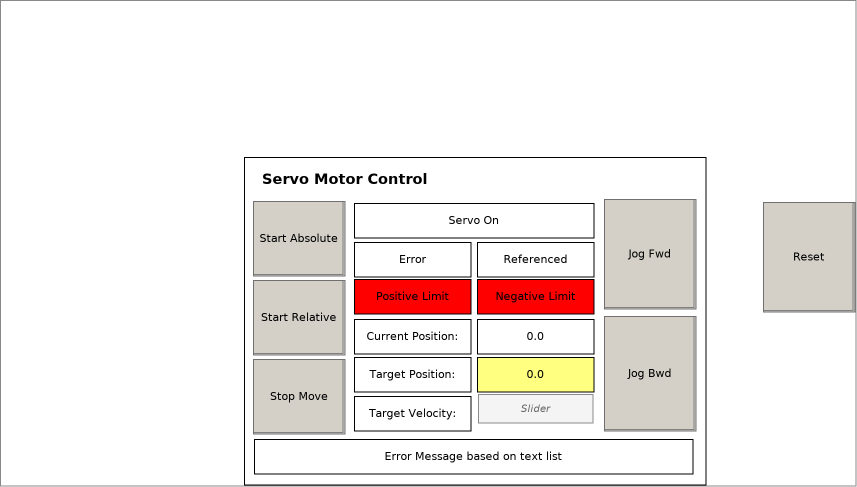
VISUALIZATION Std_BoschServo_Ctrl  // 857x487
    Rectangle (244,157 462x328)
    Button (604,199 92x110), "Jog Fwd"
        tap ER_Arm_Srv_Var.In_JogFwd
    Rectangle (354,242 117x35), "Error", colour toggle: ER_Arm_Srv_Var.Out_Error
    Rectangle (477,242 117x35), "Referenced", colour toggle: ER_Arm_Srv_Var.Out_Referenced
    Rectangle (354,279 117x35), "Positive Limit", colour toggle: ER_Arm_Srv_Var.Out_PosLimit
    Rectangle (477,279 117x35), "Negative Limit", colour toggle: ER_Arm_Srv_Var.Out_NegLimit
    Rectangle (254,439 439x35), "Error Message based on text list", text variable: MAIN.Drive1Var.Out_ErrorWord, colour toggle: ER_Arm_Srv_Var.Out_Error
    Button (604,316 92x115), "Jog Bwd"
        tap ER_Arm_Srv_Var.In_JogBwd
    Button (253,201 92x75), "Start Absolute"
        tap ER_Arm_Srv_Var.In_MoveAbs
    Rectangle (354,319 117x35), "Current Position:"
    Rectangle (354,357 117x35), "Target Position:"
    Rectangle (354,396 117x35), "Target Velocity:"
    Label (259,164 247x30), "Servo Motor Control"
    Rectangle (477,319 117x35), "0.0", text variable: MAIN.Drive1Var.Out_CurrPos, input disabled if: TRUE
    Rectangle (477,357 117x35), "0.0"
    Button (253,280 92x75), "Start Relative"
        tap ER_Arm_Srv_Var.In_MoveRel
    Rectangle (354,203 240x35), "Servo On", colour toggle: ER_Arm_Srv_Var.Out_Ready
        toggle ER_Arm_Srv_Var.In_ServoOn
    Button (763,202 92x110), "Reset"
        tap ER_Servo_Output.Reset
    Button (253,359 92x75), "Stop Move"
        tap ER_Arm_Srv_Var.In_StopMove
    Slider (478,394 115x29), variable: MAIN.Drive1Var.In_VelCmd, scale 0..200
END_VISUALIZATION

(* stored: Version 1.1.0.1, ProductVersion 3.1.4018.2
   Visu Std_BoschServo_Ctrl: Id {43a81930-7a8d-4cd3-af52-3ad929b2067b} *)
